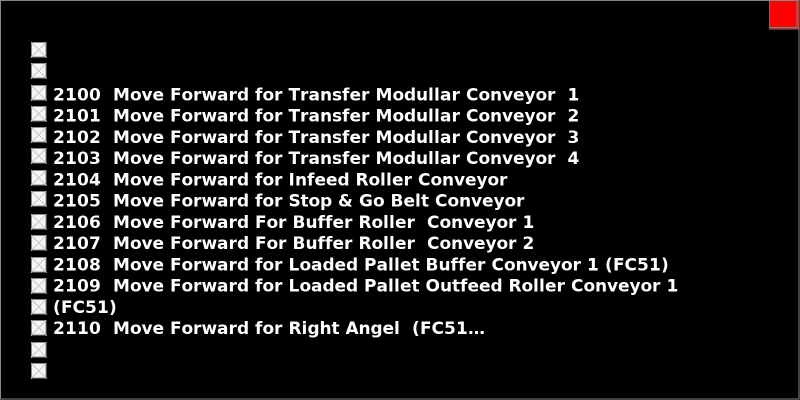
VISUALIZATION P2_DO2  // 800x400, background image 
    ImageSwitcher (31,42 15x15), variable: InputOutput_GVL.Digital_Output[17], behaviour: TOGGLE
    Label (50,16 668x391), "2100 Move Forward for Transfer Modullar Conveyor 1 2101 Move Forward for Transfer Modullar Conveyor 2 2102 Move Forward for Transfer Modullar Conveyor 3 2103 Move Forward for Transfer Modullar Conveyor 4 2104 Move Forward for Infeed Roller Conveyor 2105 Move Forward for Stop & Go Belt Conveyor 2106 Move Forward For Buffer Roller Conveyor 1 2107 Move Forward For Buffer Roller Conveyor 2 2108 Move Forward for Loaded Pallet Buffer Conveyor 1 (FC51) 2109 Move Forward for Loaded Pallet Outfeed Roller Conveyor 1 (FC51) 2110 Move Forward for Right Angel (FC51) 2111 Move Forward for Right Angel Lifter (FC51) 2112 Move Forward for Loaded Pallet Outfeed Roller Conveyor (FC51) 2113 Move Forward for Loaded Pallet Outfeed Roller Conveyor (FC51) 2114 Move Forward for Loaded Pallet Outfeed Roller Conveyor (FC51) 2115 Reset Error for All Inverter at P2, Relay"
    ImageSwitcher (31,63 15x15), variable: InputOutput_GVL.Digital_Output[18], behaviour: TOGGLE
    ImageSwitcher (31,85 15x15), variable: InputOutput_GVL.Digital_Output[19], behaviour: TOGGLE
    ImageSwitcher (31,106 15x15), variable: InputOutput_GVL.Digital_Output[20], behaviour: TOGGLE
    ImageSwitcher (31,127 15x15), variable: InputOutput_GVL.Digital_Output[21], behaviour: TOGGLE
    ImageSwitcher (31,148 15x15), variable: InputOutput_GVL.Digital_Output[22], behaviour: TOGGLE
    ImageSwitcher (31,170 15x15), variable: InputOutput_GVL.Digital_Output[23], behaviour: TOGGLE
    ImageSwitcher (31,191 15x15), variable: InputOutput_GVL.Digital_Output[24], behaviour: TOGGLE
    ImageSwitcher (31,214 15x15), variable: InputOutput_GVL.Digital_Output[25], behaviour: TOGGLE
    ImageSwitcher (31,235 15x15), variable: InputOutput_GVL.Digital_Output[26], behaviour: TOGGLE
    ImageSwitcher (31,257 15x15), variable: InputOutput_GVL.Digital_Output[27], behaviour: TOGGLE
    ImageSwitcher (31,278 15x15), variable: InputOutput_GVL.Digital_Output[28], behaviour: TOGGLE
    ImageSwitcher (31,299 15x15), variable: InputOutput_GVL.Digital_Output[29], behaviour: TOGGLE
    ImageSwitcher (31,320 15x15), variable: InputOutput_GVL.Digital_Output[30], behaviour: TOGGLE
    ImageSwitcher (31,342 15x15), variable: InputOutput_GVL.Digital_Output[31], behaviour: TOGGLE
    ImageSwitcher (31,363 15x15), variable: InputOutput_GVL.Digital_Output[32], behaviour: TOGGLE
    Button (769,-1 30x30), image: VisuSymbols.Symbols.Wrong
        OnMouseClick: CloseDialog Dialog=P2_DO2, Result=OK, NumpadKeypadSet=True
END_VISUALIZATION

(* stored: Version 1.1.0.1, ProductVersion 3.1.4024.12
   Visu P2_DO2: Id {aa1876d1-241a-426d-94ce-3ad3556dcdb2} *)
